TYPE ST_Descriptor2 :
    STRUCT
        ID    : DINT;
        Name  : STRING;
        Unit  : STRING(8);
        Value : LREAL;
    END_STRUCT
END_TYPE

(* stored: Version 1.1.0.1
   DUT ST_Descriptor2: Id {459f8359-51bb-4940-8282-2c669ca8a851} *)
